// TIA Portal V20 export
TYPE "LER_TypeFATMode_Capability"
// stored: Access Published
   STRUCT
      ProcessValue : "LER_TypeFATMode_Capability_ProcessValue";
      SetValue : "LER_TypeFATMode_Capability_SetValue";
   END_STRUCT;
END_TYPE
